% RSLogix 500 project Pruebas PID.RSS, saved by version 8.30.00.16 %
PROJECT "P1011222"    % processor: Bul.1763 MicroLogix 1100 Series B %

PROGRAM FILES
  LAD 2   10 rungs

DATA FILES
  O0 OUTPUT  6 elements
  I1 INPUT  12 elements
  S2 STATUS  66 elements
  B3 BINARY  1 elements
  T4 TIMER  1 elements
  C5 COUNTER  1 elements
  R6 CONTROL  1 elements
  N7 INTEGER  10 elements
  F8 FLOAT  9 elements
  PD9   1 elements

LADDER 2
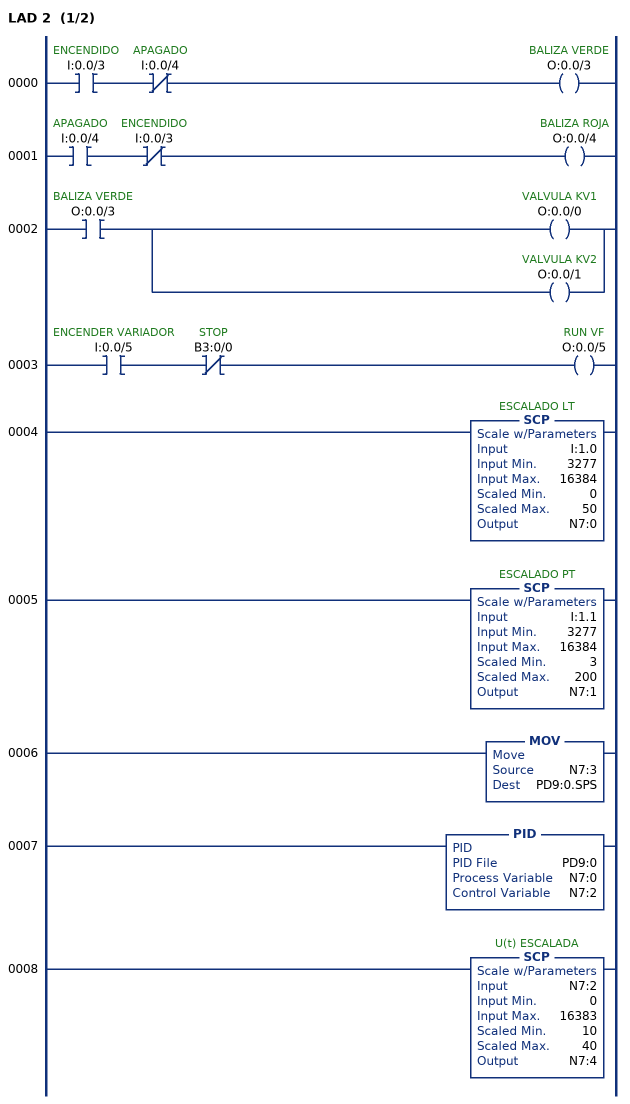
% Rung: 0 %
SOR XIC I:0.0/3 XIO I:0.0/4 OTE O:0.0/3 EOR
%   I:0.0/3  "ENCENDIDO" %
%   I:0.0/4  "APAGADO" %
%   O:0.0/3  "BALIZA VERDE" %
% Rung: 1 %
SOR XIC I:0.0/4 XIO I:0.0/3 OTE O:0.0/4 EOR
%   I:0.0/4  "APAGADO" %
%   I:0.0/3  "ENCENDIDO" %
%   O:0.0/4  "BALIZA ROJA" %
% Rung: 2 %
SOR XIC O:0.0/3 BST OTE O:0.0/0 NXB OTE O:0.0/1 BND EOR
%   O:0.0/3  "BALIZA VERDE" %
%   O:0.0/0  "VALVULA KV1" %
%   O:0.0/1  "VALVULA KV2" %
% Rung: 3 %
SOR XIC I:0.0/5 XIO B3:0/0 OTE O:0.0/5 EOR
%   I:0.0/5  "ENCENDER VARIADOR" %
%   B3:0/0  "STOP" %
%   O:0.0/5  "RUN VF" %
% Rung: 4 %
SOR SCP I:1.0 3277 16384 0 50 N7:0 EOR
%   I:1.0  "LT" %
%   N7:0  "ESCALADO LT" %
% Rung: 5 %
SOR SCP I:1.1 3277 16384 3 200 N7:1 EOR
%   I:1.1  "PT" %
%   N7:1  "ESCALADO PT" %
% Rung: 6 %
SOR MOV N7:3 PD9:0.SPS EOR
%   N7:3  "SET POINT" %
% Rung: 7 %
SOR PID PD9:0 N7:0 N7:2 EOR
%   N7:0  "ESCALADO LT" %
%   N7:2  "SALIDA PID" %
% Rung: 8 %
SOR SCP N7:2 0 16383 10 40 N7:4 EOR
%   N7:2  "SALIDA PID" %
%   N7:4  "U(t) ESCALADA" %

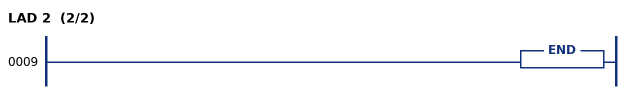
% Rung: 9 %
SOR END EOR

OTHER DOCUMENTED ADDRESSES
  F8:0  "SP"
  F8:1  "kc"
  F8:2  "ti"
  F8:3  "td"
  O:1.0  "SENAL U(t)"
  PD9:0.2  "REFERENCIA"
  PD9:0.3  "Kc"
  PD9:0.4  "Ti"
  PD9:0.5  "Td"

DATA TABLE (non-zero values as saved)
DATA N7
% N7:0 % 7 14 0 20 10 1 3 -6 -6 6
DATA F8
% F8:0 % 40 1 3 0 16384
